FUNCTION_BLOCK socketClient (* Composite Function Block Type *)
  (* Standard: 61499-2 *)
  (* Version 0.0, 2018-02-07, 4DIAC-IDE, 4DIAC-Consortium *)
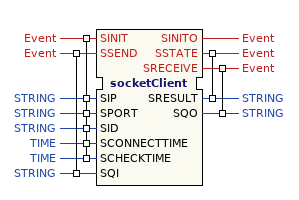
  EVENT_INPUT
    SINIT WITH SCHECKTIME, SCONNECTTIME, SID, SPORT, SIP; (* Initialization Request *)
    SSEND WITH SQI; (* Normal Execution Request *)
  END_EVENT
  EVENT_OUTPUT
    SINITO; (* Initialization Confirm *)
    SSTATE WITH SRESULT; (* Execution Confirmation *)
    SRECEIVE WITH SQO;
  END_EVENT
  VAR_INPUT
    SIP : STRING;
    SPORT : STRING;
    SID : STRING;
    SCONNECTTIME : TIME;
    SCHECKTIME : TIME;
    SQI : STRING; (* Input event qualifier *)
  END_VAR
  VAR_OUTPUT
    SRESULT : STRING;
    SQO : STRING; (* Output event qualifier *)
  END_VAR
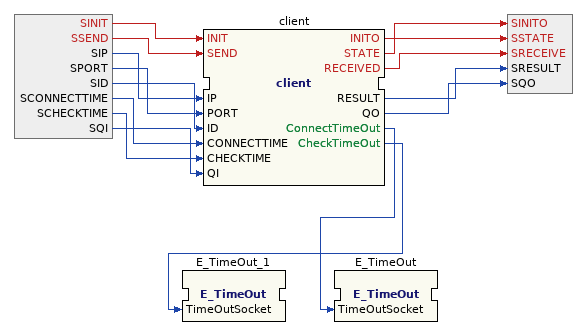
  FBS
    client : client;
    E_TimeOut : E_TimeOut;
    E_TimeOut_1 : E_TimeOut;
  END_FBS
  EVENT_CONNECTIONS
    client.RECEIVED TO SRECEIVE;
    client.STATE TO SSTATE;
    client.INITO TO SINITO;
    SSEND TO client.SEND;
    SINIT TO client.INIT;
  END_CONNECTIONS
  DATA_CONNECTIONS
    client.ConnectTimeOut TO E_TimeOut.TimeOutSocket;
    client.CheckTimeOut TO E_TimeOut_1.TimeOutSocket;
    client.QO TO SQO;
    client.RESULT TO SRESULT;
    SQI TO client.QI;
    SCHECKTIME TO client.CHECKTIME;
    SCONNECTTIME TO client.CONNECTTIME;
    SID TO client.ID;
    SPORT TO client.PORT;
    SIP TO client.IP;
  END_CONNECTIONS
END_FUNCTION_BLOCK
